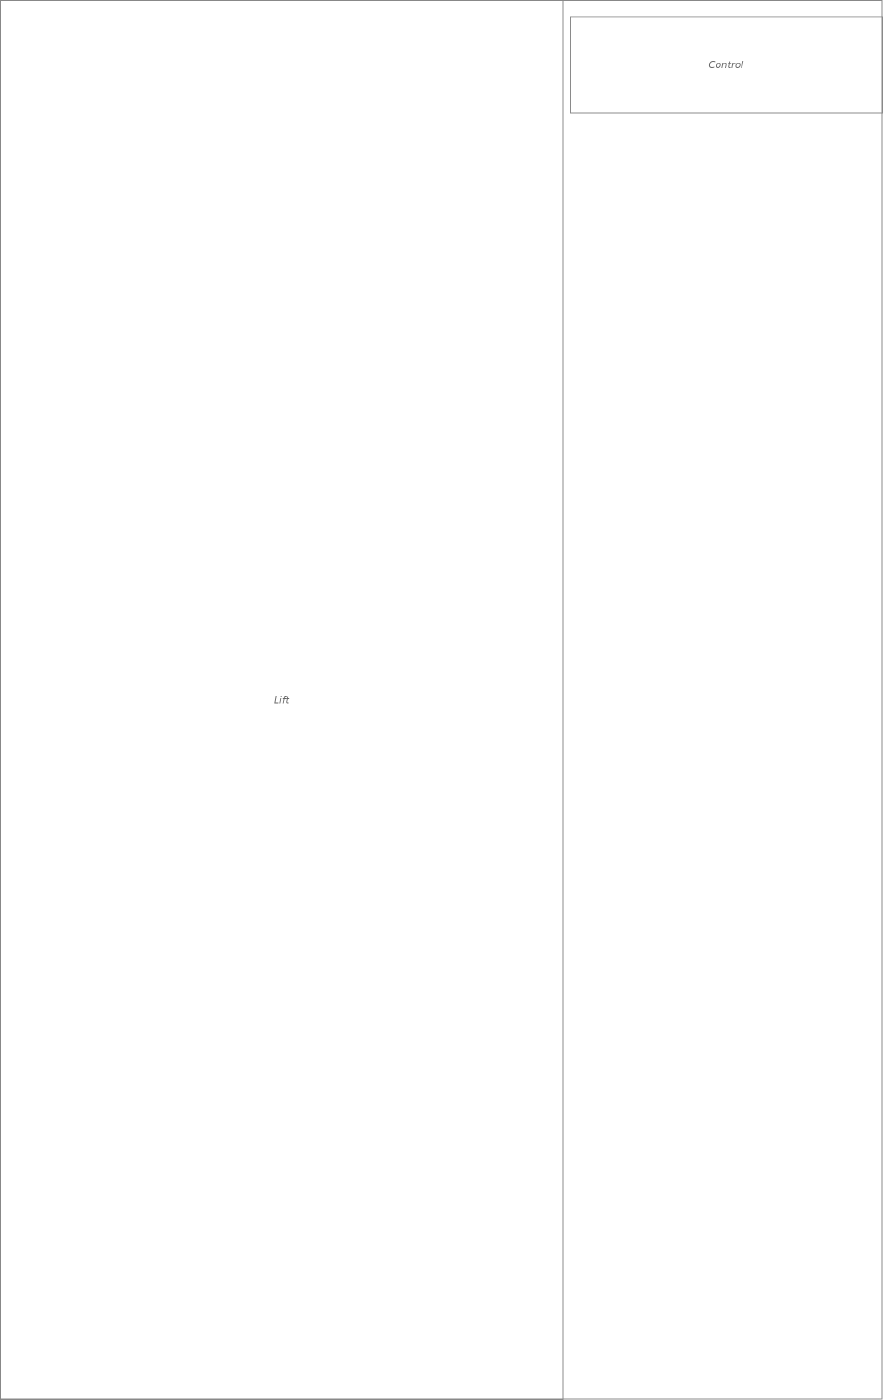
VISUALIZATION Lift_1  // 922x1461
    Frame (0,0 588x1461)
        shows Lift(Position := Visu_L1.Position_LIFT, RefSensor := Visu_L1.Control_LiftAxisReference, Color := Visu_L1.Color, Door_1_Position := Visu_L1.Door_1_Position, Door_1_M_Open := Visu_L1.Door_1_M_Open, Door_1_M_Close := Visu_L1.Door_1_M_Close, Door_2_Position := Visu_L1.Door_2_Position, Door_2_M_Open := Visu_L1.Door_2_M_Open, Door_2_M_Close := Visu_L1.Door_2_M_Close, Door_3_Position := Visu_L1.Door_3_Position, Door_3_M_Open := Visu_L1.Door_3_M_Open, Door_3_M_Close := Visu_L1.Door_3_M_Close, Door_4_Position := Visu_L1.Door_4_Position, Door_4_M_Open := Visu_L1.Door_4_M_Open, Door_4_M_Close := Visu_L1.Door_4_M_Close, Door_5_Position := Visu_L1.Door_5_Position, Door_5_M_Open := Visu_L1.Door_5_M_Open, Door_5_M_Close := Visu_L1.Door_5_M_Close, Door_6_Position := Visu_L1.Door_6_Position, Door_6_M_Open := Visu_L1.Door_6_M_Open, Door_6_M_Close := Visu_L1.Door_6_M_Close, LED_Up_1 := Visu_L1.Panel_1_Led_Up, LED_Down_1 := Visu_L1.Panel_1_Led_Down, FloorNumber_1 := Visu_L1.Panel_1_FloorNumber, BtnLed_1 := Visu_L1.Panel_1_BtnLed, Btn_1 := Visu_L1.Panel_1_Btn, LB_1 := Visu_L1.Door_1_SensorActive, LED_DoorOpen_1 := Visu_L1.Door_1_SensorOpen, LED_DoorClosed_1 := Visu_L1.Door_1_SensorClosed, LED_Up_2 := Visu_L1.Panel_2_Led_Up, LED_Down_2 := Visu_L1.Panel_2_Led_Down, FloorNumber_2 := Visu_L1.Panel_2_FloorNumber, BtnLed_2 := Visu_L1.Panel_2_BtnLed, Btn_2 := Visu_L1.Panel_2_Btn, LB_2 := Visu_L1.Door_2_SensorActive, LED_DoorOpen_2 := Visu_L1.Door_2_SensorOpen, LED_DoorClosed_2 := Visu_L1.Door_2_SensorClosed, LED_Up_3 := Visu_L1.Panel_3_Led_Up, LED_Down_3 := Visu_L1.Panel_3_Led_Down, FloorNumber_3 := Visu_L1.Panel_3_FloorNumber, BtnLed_3 := Visu_L1.Panel_3_BtnLed, Btn_3 := Visu_L1.Panel_3_Btn, LB_3 := Visu_L1.Door_3_SensorActive, LED_DoorOpen_3 := Visu_L1.Door_3_SensorOpen, LED_DoorClosed_3 := Visu_L1.Door_3_SensorClosed, LED_Up_4 := Visu_L1.Panel_4_Led_Up, LED_Down_4 := Visu_L1.Panel_4_Led_Down, FloorNumber_4 := Visu_L1.Panel_4_FloorNumber, BtnLed_4 := Visu_L1.Panel_4_BtnLed, Btn_4 := Visu_L1.Panel_4_Btn, LB_4 := Visu_L1.Door_4_SensorActive, LED_DoorOpen_4 := Visu_L1.Door_4_SensorOpen, LED_DoorClosed_4 := Visu_L1.Door_4_SensorClosed, LED_Up_5 := Visu_L1.Panel_5_Led_Up, LED_Down_5 := Visu_L1.Panel_5_Led_Down, FloorNumber_5 := Visu_L1.Panel_5_FloorNumber, BtnLed_5 := Visu_L1.Panel_5_BtnLed, Btn_5 := Visu_L1.Panel_5_Btn, LB_5 := Visu_L1.Door_5_SensorActive, LED_DoorOpen_5 := Visu_L1.Door_5_SensorOpen, LED_DoorClosed_5 := Visu_L1.Door_5_SensorClosed, LED_Up_6 := Visu_L1.Panel_6_Led_Up, LED_Down_6 := Visu_L1.Panel_6_Led_Down, FloorNumber_6 := Visu_L1.Panel_6_FloorNumber, BtnLed_6 := Visu_L1.Panel_6_BtnLed, Btn_6 := Visu_L1.Panel_6_Btn, LB_6 := Visu_L1.Door_6_SensorActive, LED_DoorOpen_6 := Visu_L1.Door_6_SensorOpen, LED_DoorClosed_6 := Visu_L1.Door_6_SensorClosed)
    Frame (595,17 327x101)
        shows Control(LED_Blue := Visu_L1.Control_LED_Blue, LED_Red := Visu_L1.Control_LED_Red, LED_White := Visu_L1.Control_LED_White, LED_Yellow := Visu_L1.Control_LED_Yellow, Start := Visu_L1.Control_Start, Reset := Visu_L1.Control_Reset, State := Visu_L1.Control_State)
END_VISUALIZATION

(* stored: Version 1.1.0.1
   Visu Lift_1: Id {a365684b-66a7-4bd1-8225-e4c71101bd2d} *)
